(* Schneider Machine Expert - Basic project outputs as inputs, file version 1.9.0.0 *)
(* ProjectInformations: Name=New project *)

HARDWARE
  Cpu 0: TM221CE16R
  EthernetConfiguration: NetworkName=M221, IpAllocationMode=FixedAddress, IpAddress=0.0.0.0, SubnetMask=0.0.0.0
  SerialLineConfiguration: Baud=Baud19200, Parity=ParityEven, DataBits=DataBits8, StopBits=StopBits1, PhysicalMedium=PhysicalMediumRs485, TransmissionMode=TransmissionModeModbusRtu, SlaveId=1, Addressing=SlaveAddressing
  MastTask: UsePeriodScanMode=false, PeriodScan=100
  FastTask: Period=255
  CpuBehavior: StartingMode=StartAsPreviousState, AutoSaveRamOnEeprom=true, WatchdogPeriod=250

SYMBOLS  (address, symbol, comment, settings)

POU New POU
  (* SectionNumber=1 *)

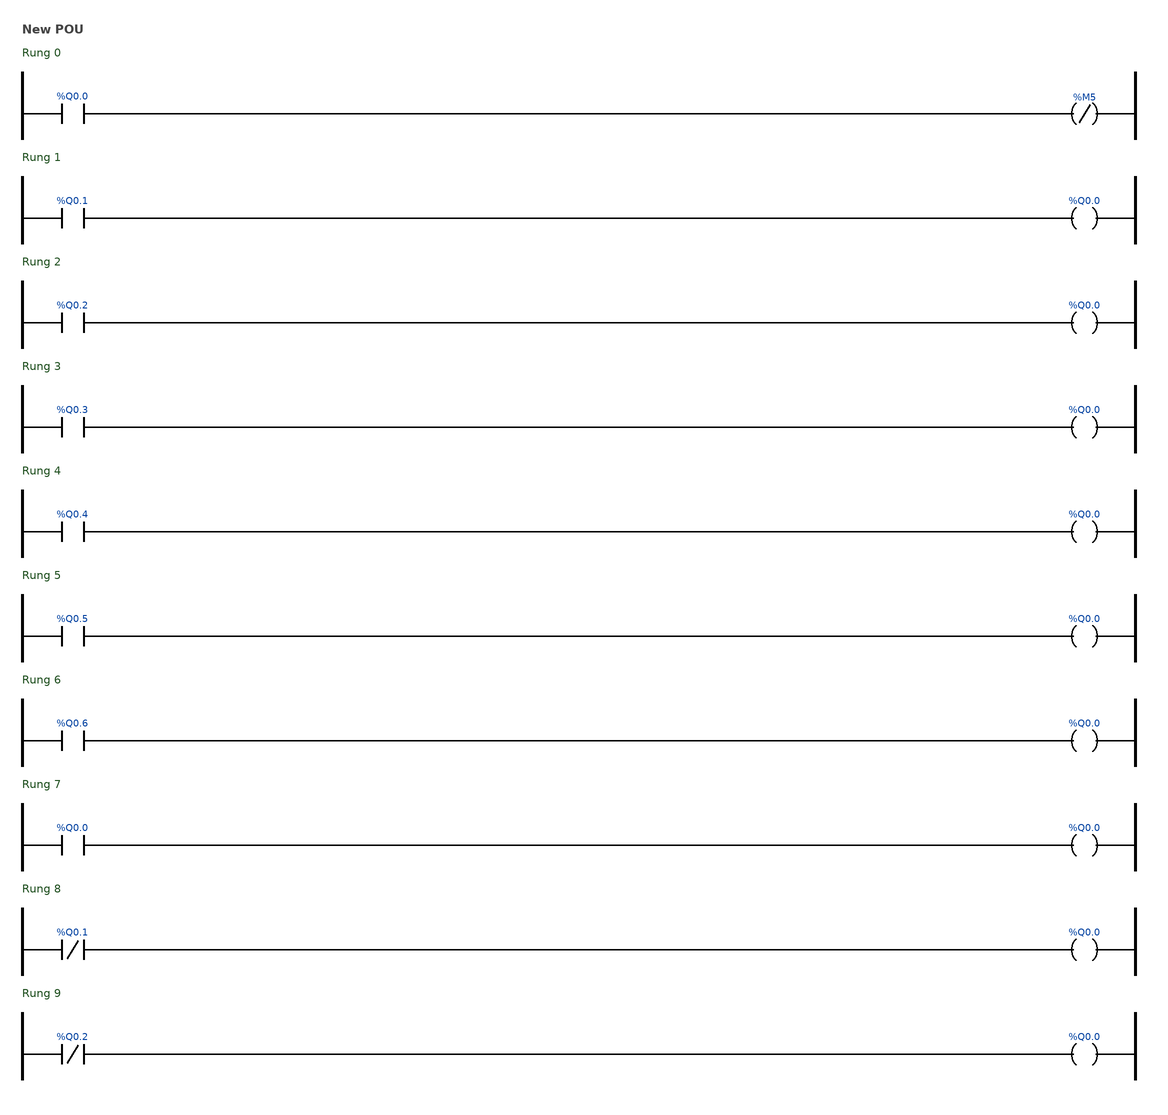

// Rung 0
  LD %Q0.0
  STN %M5
  // as ST:
  //   %M5 := NOT %Q0.0;

// Rung 1
  LD %Q0.1
  ST %Q0.0
  // as ST:
  //   %Q0.0 := %Q0.1;

// Rung 2
  LD %Q0.2
  ST %Q0.0
  // as ST:
  //   %Q0.0 := %Q0.2;

// Rung 3
  LD %Q0.3
  ST %Q0.0
  // as ST:
  //   %Q0.0 := %Q0.3;

// Rung 4
  LD %Q0.4
  ST %Q0.0
  // as ST:
  //   %Q0.0 := %Q0.4;

// Rung 5
  LD %Q0.5
  ST %Q0.0
  // as ST:
  //   %Q0.0 := %Q0.5;

// Rung 6
  LD %Q0.6
  ST %Q0.0
  // as ST:
  //   %Q0.0 := %Q0.6;

// Rung 7
  LD %Q0.0
  ST %Q0.0
  // as ST:
  //   %Q0.0 := %Q0.0;

// Rung 8
  LDN %Q0.1
  ST %Q0.0
  // as ST:
  //   %Q0.0 := NOT %Q0.1;

// Rung 9
  LDN %Q0.2
  ST %Q0.0
  // as ST:
  //   %Q0.0 := NOT %Q0.2;

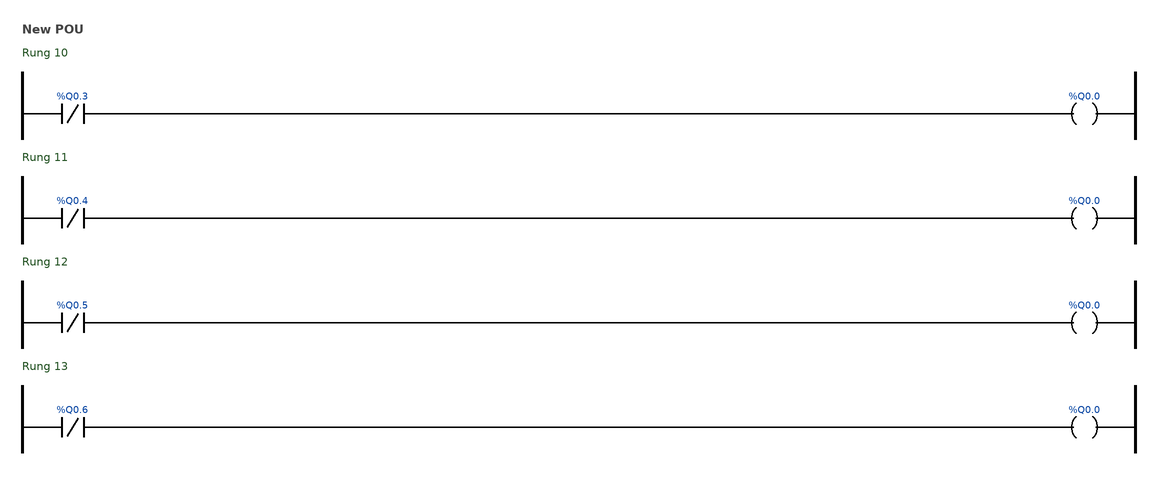

// Rung 10
  LDN %Q0.3
  ST %Q0.0
  // as ST:
  //   %Q0.0 := NOT %Q0.3;

// Rung 11
  LDN %Q0.4
  ST %Q0.0
  // as ST:
  //   %Q0.0 := NOT %Q0.4;

// Rung 12
  LDN %Q0.5
  ST %Q0.0
  // as ST:
  //   %Q0.0 := NOT %Q0.5;

// Rung 13
  LDN %Q0.6
  ST %Q0.0
  // as ST:
  //   %Q0.0 := NOT %Q0.6;
